{attribute 'GeneratedUsingTerminal: EP3204-0002-0021'}
{attribute addProperty BoxType "EP3204-0002-0021"}
{attribute addProperty Id "RTD_RTDInputs_Channel_1AT %I*AI_Standard_Channel_4A3944819RTD_RTDInputs_Channel_2AT %I*AI_Standard_Channel_4A3944819RTD_RTDInputs_Channel_3AT %I*AI_Standard_Channel_4A3944819RTD_RTDInputs_Channel_4AT %I*AI_Standard_Channel_4A3944819WcStateAT %I*WcState_9091E0EB2InfoDataAT %I*InfoData_94A18F5E2"}
{attribute addProperty CRC "1597822688"}
{attribute addProperty Size "40"}
TYPE EP3204_5F3CD6E0 EXTENDS EtcSlaveTerminalBase_947E5A46 :
STRUCT
	{attribute addProperty Name "RTD_RTDInputs_Channel_1"}
	RTD_RTDInputs_Channel_1 : AI_Standard_Channel_4A394481;
	{attribute addProperty Name "RTD_RTDInputs_Channel_2"}
	RTD_RTDInputs_Channel_2 : AI_Standard_Channel_4A394481;
	{attribute addProperty Name "RTD_RTDInputs_Channel_3"}
	RTD_RTDInputs_Channel_3 : AI_Standard_Channel_4A394481;
	{attribute addProperty Name "RTD_RTDInputs_Channel_4"}
	RTD_RTDInputs_Channel_4 : AI_Standard_Channel_4A394481;
	{attribute addProperty Name "WcState"}
	WcState : WcState_9091E0EB;
	{attribute addProperty Name "InfoData"}
	InfoData : InfoData_94A18F5E;
END_STRUCT
END_TYPE

(* stored: Version 1.2.0.0, ProductVersion 3.1.4024.9
   DUT EP3204_5F3CD6E0: Id {a9e160e8-a7be-43a9-8a65-2c9d020a3da9} *)
